INTERFACE I_DigitalSensor

PROPERTY P_FallingEdge : BOOL
GET
END_GET
END_PROPERTY

PROPERTY P_InvertLogic : BOOL
GET
END_GET
SET
END_SET
END_PROPERTY

PROPERTY P_IsActive : BOOL
GET
END_GET
END_PROPERTY

PROPERTY P_RisingEdge : BOOL
GET
END_GET
END_PROPERTY

END_INTERFACE

(* stored: Version 1.1.0.1
   Itf I_DigitalSensor: Id {4a0fb15b-571c-49ee-a291-a7cb4ebc0888}
   Property P_FallingEdge: Id {cca12828-8794-4bae-8f80-a7b224b9dd10}
   Get Get: Id {a6bfdde5-4376-4b00-a7ff-b86746c91b0c}
   Property P_InvertLogic: Id {be3a0c06-e840-4370-b33b-386d2694528b}
   Get Get: Id {2fe223f1-6213-48f1-98bd-779c84b2846c}
   Set Set: Id {71d3608d-d82c-4aba-88b6-a38bfff55f6d}
   Property P_IsActive: Id {838e7c94-ac81-4e1c-b22b-1bdd97939a7f}
   Get Get: Id {161b89e0-3288-44c4-909b-777792fb2ee5}
   Property P_RisingEdge: Id {f52a9598-e36f-4892-97b1-79ba6c72a93d}
   Get Get: Id {c02428f4-e925-4cf0-92c9-d7a48d48423b} *)
